{attribute 'qualified_only'}
{attribute 'strict'}
TYPE E_ControlBox :
(
	VirtualControlBox,
	RealControlBox
);
END_TYPE

(* stored: Version 1.1.0.1, ProductVersion 3.1.4024.12
   DUT E_ControlBox: Id {6fc44080-44ea-4649-9e9d-2d97c55e4109} *)
